// TIA Portal project "机械臂控制" (V15.1)

(* hardware
DEVICE "S7-1200 station_1"  S7-1200 Station
   slot 0: "Rack_0"  S7-1200 Rack  Rack  V1.0
   slot 1: "PLC_1"  CPU 1215C DC/DC/DC  6ES7 215-1AG40-0XB0  V4.2
*)

// ===== PLC "PLC_1"  CPU 1215C DC/DC/DC =====

VAR_GLOBAL   // PLC tag table "默认变量表"
   "Tag_1" AT %I0.0 : Bool;
   "Tag_2" AT %I0.1 : Bool;
   "Tag_3" AT %M1.0 : Bool;
   "Tag_4" AT %MD2 : DWord;
   "Tag_5" AT %MD3 : DWord;
   "Tag_6" AT %M1.1 : Bool;
   "Tag_7" AT %M1.2 : Bool;
   "Tag_8" AT %M1.3 : Bool;
   "Tag_9" AT %MD4 : DWord;
   "Tag_10" AT %M0.0 : Bool;
   "Tag_11" AT %M1.4 : Bool;
   "Tag_12" AT %M1.5 : Bool;
   "Tag_13" AT %M1.6 : Bool;
   "Tag_14" AT %M1.7 : Bool;
   "Tag_15" AT %M2.0 : Bool;
   "Tag_16" AT %M2.1 : Bool;
   "Tag_17" AT %M2.2 : Bool;
   "Tag_18" AT %M2.3 : Bool;
   "Tag_19" AT %M2.4 : Bool;
   "Tag_20" AT %Q0.5 : Bool;
   "Tag_21" AT %Q0.1 : Bool;
   "Tag_22" AT %Q0.3 : Bool;
END_VAR

// folder: System blocks/Program resources

DATA_BLOCK "IEC_Timer_0_DB"   // DB4
{ S7_Optimized_Access := 'TRUE' }
AUTHOR : Simatic
FAMILY : IEC
NAME : IEC_TMR
VERSION : 1.0
// stored: InstanceOfName IEC_TIMER
"IEC_TIMER"
BEGIN
END_DATA_BLOCK

DATA_BLOCK "IEC_Timer_0_DB_1"   // DB5
{ S7_Optimized_Access := 'TRUE' }
AUTHOR : Simatic
FAMILY : IEC
NAME : IEC_TMR
VERSION : 1.0
// stored: InstanceOfName IEC_TIMER
"IEC_TIMER"
BEGIN
END_DATA_BLOCK

DATA_BLOCK "IEC_Timer_0_DB_2"   // DB6
{ S7_Optimized_Access := 'TRUE' }
AUTHOR : Simatic
FAMILY : IEC
NAME : IEC_TMR
VERSION : 1.0
// stored: InstanceOfName IEC_TIMER
"IEC_TIMER"
BEGIN
END_DATA_BLOCK

DATA_BLOCK "IEC_Timer_0_DB_3"   // DB7
{ S7_Optimized_Access := 'TRUE' }
AUTHOR : Simatic
FAMILY : IEC
NAME : IEC_TMR
VERSION : 1.0
// stored: InstanceOfName IEC_TIMER
"IEC_TIMER"
BEGIN
END_DATA_BLOCK

// folder: (top level)

ORGANIZATION_BLOCK "Main"   // OB1, LAD, ProgramCycle
TITLE = "Main Program Sweep (Cycle)"
{ S7_Optimized_Access := 'TRUE' }
VERSION : 0.1
   VAR_INPUT
      Initial_Call : Bool;   // Initial call of this OB
      Remanence : Bool;   // =True, if remanent data are available
   END_VAR
   VAR_TEMP   // added for the SCL form of the ladder/FBD networks
      _w1 : Bool;
      _w2 : Bool;
      _w3 : Bool;
      _w4 : Bool;
      _w5 : Bool;
      _w6 : Bool;
      _w7 : Bool;
      _w8 : Bool;
      _w9 : Bool;
   END_VAR
BEGIN

REGION Network 1
   // 起动
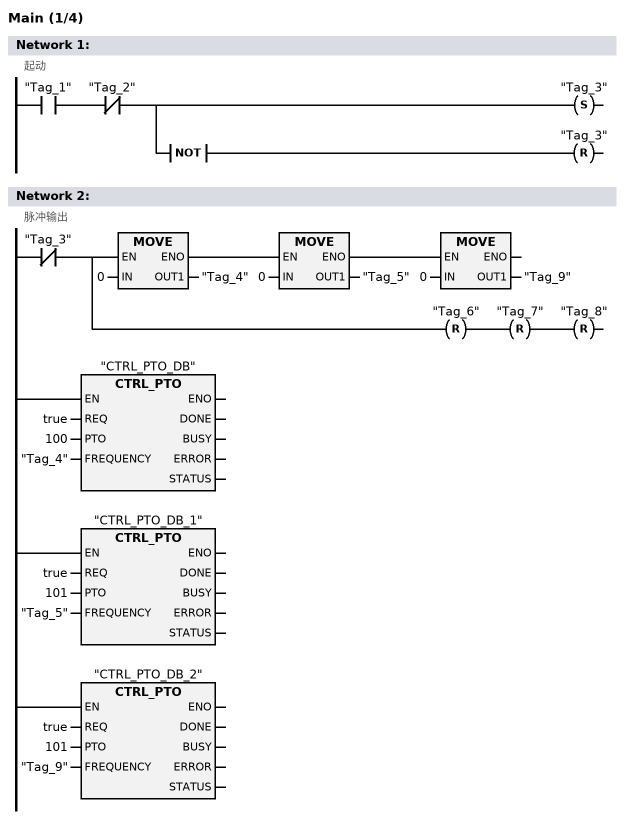
   RUNG wire#powerrail
      Contact( "Tag_1" )
      I_Contact( "Tag_2" )
      wire#w1
      S_Coil( "Tag_3" )
   END_RUNG
   RUNG wire#w1
      Not()
      R_Coil( "Tag_3" )
   END_RUNG
   // the same network as SCL:
   #_w1 := "Tag_1" AND NOT "Tag_2";
   IF #_w1 THEN "Tag_3" := TRUE; END_IF;
   IF NOT #_w1 THEN "Tag_3" := FALSE; END_IF;
END_REGION

REGION Network 2
   // 脉冲输出
   IF NOT "Tag_3" THEN
       "Tag_4" := 0;
       "Tag_5" := 0;
       "Tag_9" := 0;
       "Tag_6" := FALSE;
       "Tag_7" := FALSE;
       "Tag_8" := FALSE;
   END_IF;
   "CTRL_PTO_DB"(REQ := true, PTO := 100, FREQUENCY := "Tag_4");   // CTRL_PTO
   "CTRL_PTO_DB_1"(REQ := true, PTO := 101, FREQUENCY := "Tag_5");   // CTRL_PTO
   "CTRL_PTO_DB_2"(REQ := true, PTO := 101, FREQUENCY := "Tag_9");   // CTRL_PTO
END_REGION

REGION Network 3
   // 加速、匀速、减速
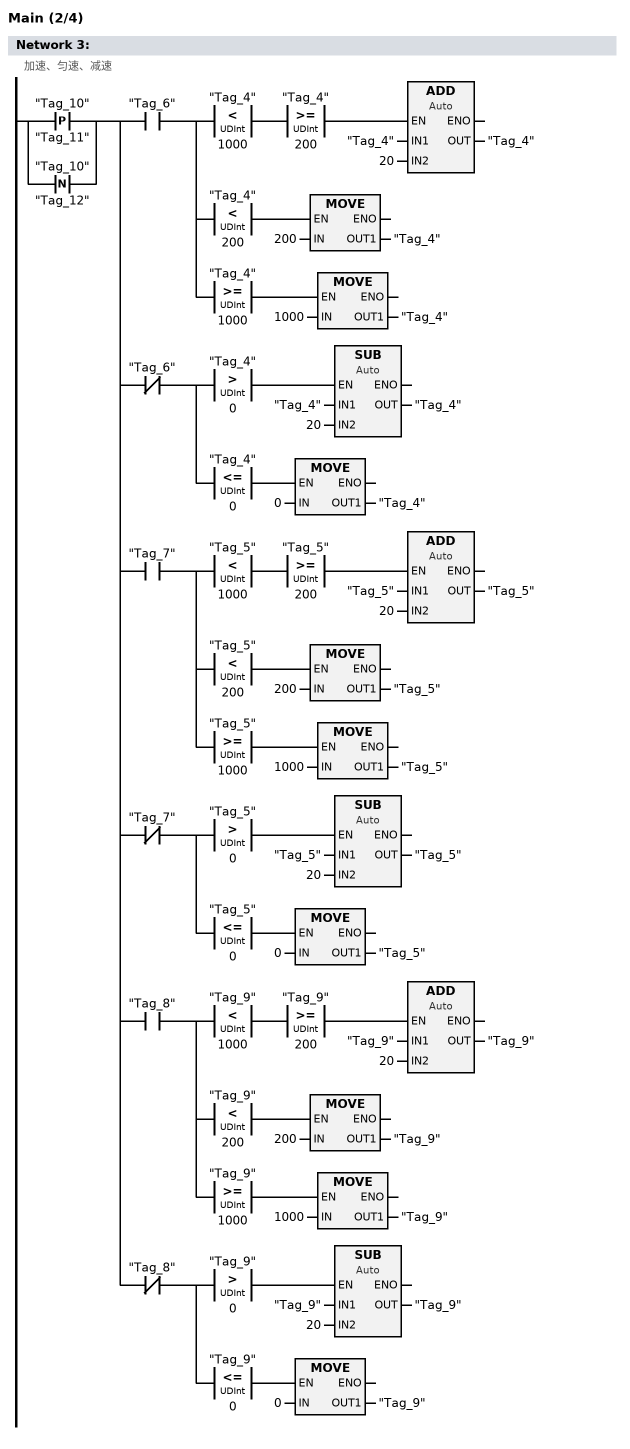
   RUNG wire#powerrail
      P_Contact(operand := "Tag_10", bit := "Tag_11")
      wire#w1
      Contact( "Tag_6" )
      wire#w2
      { S7_Templates := "SrcType := UDInt" } LT_Contact(in1 := "Tag_4", in2 := 1000)
      { S7_Templates := "SrcType := UDInt" } GE_Contact(in1 := "Tag_4", in2 := 200)
      Add(in1 := "Tag_4", in2 := 20, out => "Tag_4")
   END_RUNG
   RUNG wire#powerrail
      N_Contact(operand := "Tag_10", bit := "Tag_12")
   END_RUNG wire#w1
   RUNG wire#w2
      { S7_Templates := "SrcType := UDInt" } LT_Contact(in1 := "Tag_4", in2 := 200)
      Move(in := 200, out1 => "Tag_4")
   END_RUNG
   RUNG wire#w2
      { S7_Templates := "SrcType := UDInt" } GE_Contact(in1 := "Tag_4", in2 := 1000)
      Move(in := 1000, out1 => "Tag_4")
   END_RUNG
   RUNG wire#w1
      I_Contact( "Tag_6" )
      wire#w3
      { S7_Templates := "SrcType := UDInt" } GT_Contact(in1 := "Tag_4", in2 := 0)
      Sub(in1 := "Tag_4", in2 := 20, out => "Tag_4")
   END_RUNG
   RUNG wire#w3
      { S7_Templates := "SrcType := UDInt" } LE_Contact(in1 := "Tag_4", in2 := 0)
      Move(in := 0, out1 => "Tag_4")
   END_RUNG
   RUNG wire#w1
      Contact( "Tag_7" )
      wire#w4
      { S7_Templates := "SrcType := UDInt" } LT_Contact(in1 := "Tag_5", in2 := 1000)
      { S7_Templates := "SrcType := UDInt" } GE_Contact(in1 := "Tag_5", in2 := 200)
      Add(in1 := "Tag_5", in2 := 20, out => "Tag_5")
   END_RUNG
   RUNG wire#w4
      { S7_Templates := "SrcType := UDInt" } LT_Contact(in1 := "Tag_5", in2 := 200)
      Move(in := 200, out1 => "Tag_5")
   END_RUNG
   RUNG wire#w4
      { S7_Templates := "SrcType := UDInt" } GE_Contact(in1 := "Tag_5", in2 := 1000)
      Move(in := 1000, out1 => "Tag_5")
   END_RUNG
   RUNG wire#w1
      I_Contact( "Tag_7" )
      wire#w5
      { S7_Templates := "SrcType := UDInt" } GT_Contact(in1 := "Tag_5", in2 := 0)
      Sub(in1 := "Tag_5", in2 := 20, out => "Tag_5")
   END_RUNG
   RUNG wire#w5
      { S7_Templates := "SrcType := UDInt" } LE_Contact(in1 := "Tag_5", in2 := 0)
      Move(in := 0, out1 => "Tag_5")
   END_RUNG
   RUNG wire#w1
      Contact( "Tag_8" )
      wire#w6
      { S7_Templates := "SrcType := UDInt" } LT_Contact(in1 := "Tag_9", in2 := 1000)
      { S7_Templates := "SrcType := UDInt" } GE_Contact(in1 := "Tag_9", in2 := 200)
      Add(in1 := "Tag_9", in2 := 20, out => "Tag_9")
   END_RUNG
   RUNG wire#w6
      { S7_Templates := "SrcType := UDInt" } LT_Contact(in1 := "Tag_9", in2 := 200)
      Move(in := 200, out1 => "Tag_9")
   END_RUNG
   RUNG wire#w6
      { S7_Templates := "SrcType := UDInt" } GE_Contact(in1 := "Tag_9", in2 := 1000)
      Move(in := 1000, out1 => "Tag_9")
   END_RUNG
   RUNG wire#w1
      I_Contact( "Tag_8" )
      wire#w7
      { S7_Templates := "SrcType := UDInt" } GT_Contact(in1 := "Tag_9", in2 := 0)
      Sub(in1 := "Tag_9", in2 := 20, out => "Tag_9")
   END_RUNG
   RUNG wire#w7
      { S7_Templates := "SrcType := UDInt" } LE_Contact(in1 := "Tag_9", in2 := 0)
      Move(in := 0, out1 => "Tag_9")
   END_RUNG
   // the same network as SCL:
   #_w1 := "Tag_10" AND NOT "Tag_11";   // rising edge of "Tag_10"
   "Tag_11" := "Tag_10";
   #_w2 := NOT "Tag_10" AND "Tag_12";   // falling edge of "Tag_10"
   "Tag_12" := "Tag_10";
   #_w3 := #_w1 OR #_w2;
   #_w4 := #_w3 AND "Tag_6";
   IF #_w4 AND ("Tag_4" < 1000) AND ("Tag_4" >= 200) THEN "Tag_4" := "Tag_4" + 20; END_IF;
   IF #_w4 AND ("Tag_4" < 200) THEN "Tag_4" := 200; END_IF;
   IF #_w4 AND ("Tag_4" >= 1000) THEN "Tag_4" := 1000; END_IF;
   #_w5 := #_w3 AND NOT "Tag_6";
   IF #_w5 AND ("Tag_4" > 0) THEN "Tag_4" := "Tag_4" - 20; END_IF;
   IF #_w5 AND ("Tag_4" <= 0) THEN "Tag_4" := 0; END_IF;
   #_w6 := #_w3 AND "Tag_7";
   IF #_w6 AND ("Tag_5" < 1000) AND ("Tag_5" >= 200) THEN "Tag_5" := "Tag_5" + 20; END_IF;
   IF #_w6 AND ("Tag_5" < 200) THEN "Tag_5" := 200; END_IF;
   IF #_w6 AND ("Tag_5" >= 1000) THEN "Tag_5" := 1000; END_IF;
   #_w7 := #_w3 AND NOT "Tag_7";
   IF #_w7 AND ("Tag_5" > 0) THEN "Tag_5" := "Tag_5" - 20; END_IF;
   IF #_w7 AND ("Tag_5" <= 0) THEN "Tag_5" := 0; END_IF;
   #_w8 := #_w3 AND "Tag_8";
   IF #_w8 AND ("Tag_9" < 1000) AND ("Tag_9" >= 200) THEN "Tag_9" := "Tag_9" + 20; END_IF;
   IF #_w8 AND ("Tag_9" < 200) THEN "Tag_9" := 200; END_IF;
   IF #_w8 AND ("Tag_9" >= 1000) THEN "Tag_9" := 1000; END_IF;
   #_w9 := #_w3 AND NOT "Tag_8";
   IF #_w9 AND ("Tag_9" > 0) THEN "Tag_9" := "Tag_9" - 20; END_IF;
   IF #_w9 AND ("Tag_9" <= 0) THEN "Tag_9" := 0; END_IF;
END_REGION

REGION Network 4
   // 自动运行
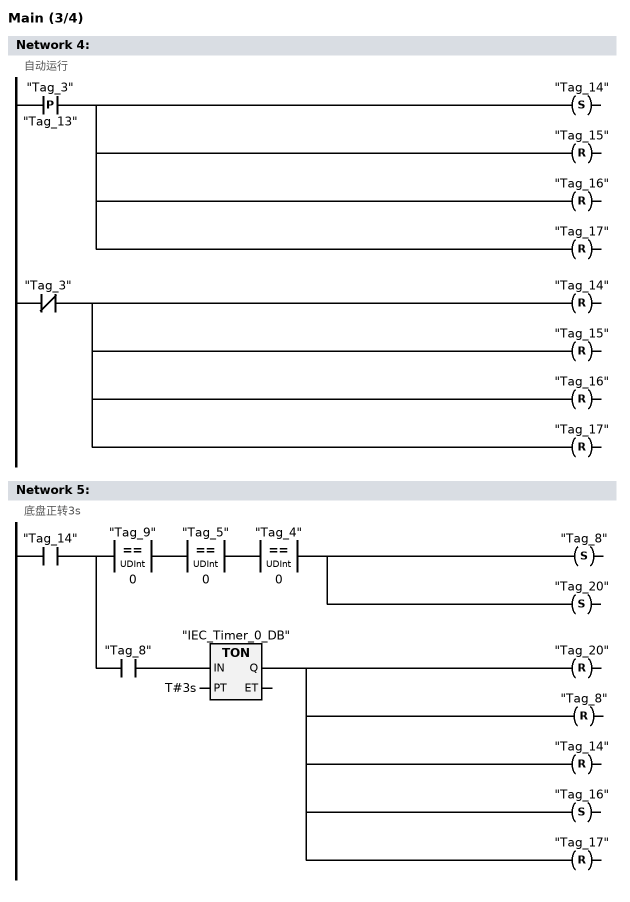
   RUNG wire#powerrail
      P_Contact(operand := "Tag_3", bit := "Tag_13")
      wire#w1
      S_Coil( "Tag_14" )
   END_RUNG
   RUNG wire#w1
      R_Coil( "Tag_15" )
   END_RUNG
   RUNG wire#w1
      R_Coil( "Tag_16" )
   END_RUNG
   RUNG wire#w1
      R_Coil( "Tag_17" )
   END_RUNG
   RUNG wire#powerrail
      I_Contact( "Tag_3" )
      wire#w2
      R_Coil( "Tag_14" )
   END_RUNG
   RUNG wire#w2
      R_Coil( "Tag_15" )
   END_RUNG
   RUNG wire#w2
      R_Coil( "Tag_16" )
   END_RUNG
   RUNG wire#w2
      R_Coil( "Tag_17" )
   END_RUNG
   // the same network as SCL:
   #_w1 := "Tag_3" AND NOT "Tag_13";   // rising edge of "Tag_3"
   "Tag_13" := "Tag_3";
   IF #_w1 THEN
       "Tag_14" := TRUE;
       "Tag_15" := FALSE;
       "Tag_16" := FALSE;
       "Tag_17" := FALSE;
   END_IF;
   IF NOT "Tag_3" THEN
       "Tag_14" := FALSE;
       "Tag_15" := FALSE;
       "Tag_16" := FALSE;
       "Tag_17" := FALSE;
   END_IF;
END_REGION

REGION Network 5
   // 底盘正转3s
   IF "Tag_14" AND ("Tag_9" = 0) AND ("Tag_5" = 0) AND ("Tag_4" = 0) THEN
       "Tag_8" := TRUE;
       "Tag_20" := TRUE;
   END_IF;
   "IEC_Timer_0_DB".TON(IN := "Tag_14" AND "Tag_8", PT := T#3s);
   IF "IEC_Timer_0_DB".Q THEN
       "Tag_20" := FALSE;
       "Tag_8" := FALSE;
       "Tag_14" := FALSE;
       "Tag_16" := TRUE;
       "Tag_17" := FALSE;
   END_IF;
END_REGION

REGION Network 6
   // 大小臂正转5s后反转5s
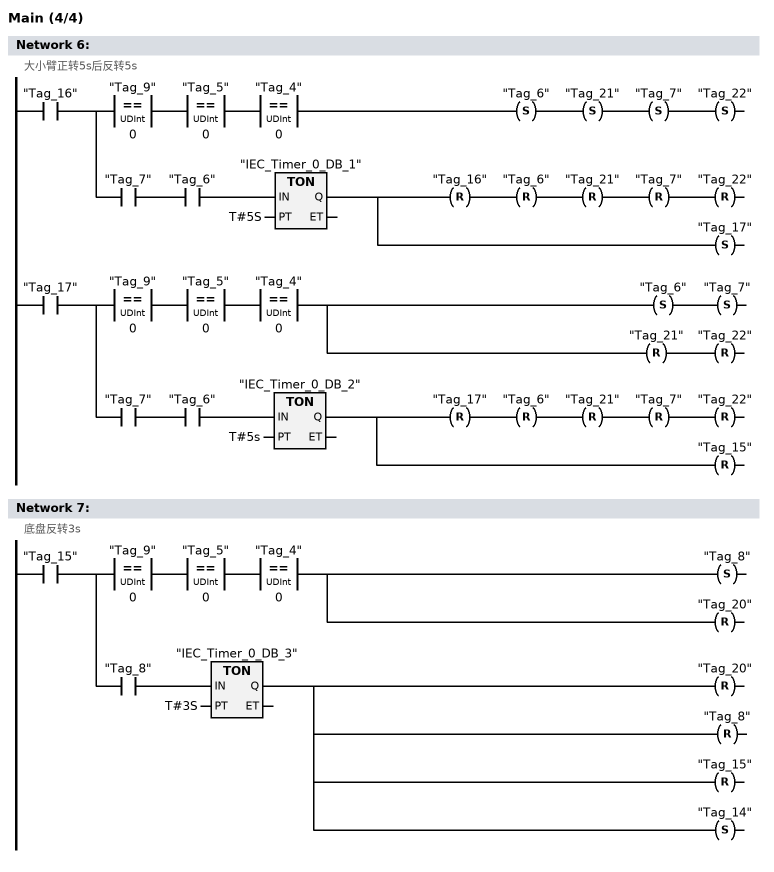
   IF "Tag_16" AND ("Tag_9" = 0) AND ("Tag_5" = 0) AND ("Tag_4" = 0) THEN
       "Tag_6" := TRUE;
       "Tag_21" := TRUE;
       "Tag_7" := TRUE;
       "Tag_22" := TRUE;
   END_IF;
   "IEC_Timer_0_DB_1".TON(IN := "Tag_16" AND "Tag_7" AND "Tag_6", PT := T#5S);
   IF "IEC_Timer_0_DB_1".Q THEN
       "Tag_16" := FALSE;
       "Tag_6" := FALSE;
       "Tag_21" := FALSE;
       "Tag_7" := FALSE;
       "Tag_22" := FALSE;
       "Tag_17" := TRUE;
   END_IF;
   IF "Tag_17" AND ("Tag_9" = 0) AND ("Tag_5" = 0) AND ("Tag_4" = 0) THEN
       "Tag_6" := TRUE;
       "Tag_7" := TRUE;
       "Tag_21" := FALSE;
       "Tag_22" := FALSE;
   END_IF;
   "IEC_Timer_0_DB_2".TON(IN := "Tag_17" AND "Tag_7" AND "Tag_6", PT := T#5s);
   IF "IEC_Timer_0_DB_2".Q THEN
       "Tag_17" := FALSE;
       "Tag_6" := FALSE;
       "Tag_21" := FALSE;
       "Tag_7" := FALSE;
       "Tag_22" := FALSE;
       "Tag_15" := FALSE;
   END_IF;
END_REGION

REGION Network 7
   // 底盘反转3s
   IF "Tag_15" AND ("Tag_9" = 0) AND ("Tag_5" = 0) AND ("Tag_4" = 0) THEN
       "Tag_8" := TRUE;
       "Tag_20" := FALSE;
   END_IF;
   "IEC_Timer_0_DB_3".TON(IN := "Tag_15" AND "Tag_8", PT := T#3S);
   IF "IEC_Timer_0_DB_3".Q THEN
       "Tag_20" := FALSE;
       "Tag_8" := FALSE;
       "Tag_15" := FALSE;
       "Tag_14" := TRUE;
   END_IF;
END_REGION
END_ORGANIZATION_BLOCK